INTERFACE I_RpcProxy

PROPERTY bIsConfigured : BOOL
GET
END_GET
END_PROPERTY

METHOD GetVerificationResult : HRESULT

VAR_OUTPUT
	stResult : ST_VerificationResult;
END_VAR
END_METHOD

PROPERTY itfTestFrameWorkAdapter :  I_TestFrameWorkAdapter
GET
END_GET
SET
END_SET
END_PROPERTY

METHOD Verify : HRESULT
VAR_INPUT CONSTANT
	sToVerify	: REFERENCE TO T_VerifyContent;
END_VAR
END_METHOD

END_INTERFACE

(* stored: Version 1.1.0.1, ProductVersion 3.1.4026.18
   Itf I_RpcProxy: Id {3c923e29-1b12-4fb6-918d-7d40a223d3a1}
   Property bIsConfigured: Id {6b71f334-0487-4b78-b6c4-19f75fda71e2}
   Get Get: Id {b19647cb-c647-46f6-a26a-f86ef22837c5}
   Method GetVerificationResult: Id {8c21d341-bad1-455d-9cad-76e4aed1c398}
   Property itfTestFrameWorkAdapter: Id {3cc412ee-5500-45a0-813f-576cd1d9ffe3}
   Get Get: Id {02bd8883-b639-4619-b8d8-ab745a2fcaa2}
   Set Set: Id {3a99c542-237f-4bcf-ba74-d6665c8c0976}
   Method Verify: Id {11e40880-5fa3-4b04-ac89-634a6cfbe115} *)
